TYPE ST001_ProcessData EXTENDS TcoData.TcoEntity:
STRUCT
	PressingTime : TIME;
END_STRUCT
END_TYPE

(* stored: Version 1.1.0.1
   DUT ST001_ProcessData: Id {e8ba0c5f-1502-08c8-06c0-eb4e9bcba2df} *)
